FUNCTION_BLOCK FB_FallibleSTRINGMock IMPLEMENTS I_FallibleSTRING
VAR
    bError : BOOL;
    sErrorMsg : T_MaxString;
    sVal : STRING;
END_VAR


METHOD ClearError

bError := FALSE;
sErrorMsg := '';
END_METHOD


METHOD GetError : BOOL

GetError := THIS^.bError;
END_METHOD


METHOD GetErrorMsg : T_MaxString

GetErrorMsg := sErrorMsg;
END_METHOD


METHOD PUBLIC SetError
VAR_INPUT
    sMsg : T_MaxString;
END_VAR

THIS^.bError := TRUE;
END_METHOD


PROPERTY Val : STRING
GET

Val := THIS^.sVal;
END_GET
SET

THIS^.sVal := Val;
END_SET
END_PROPERTY

END_FUNCTION_BLOCK

(* stored: Version 1.1.0.1
   POU FB_FallibleSTRINGMock: Id {a03a76bb-b88e-4cb0-a83d-4c8c1047d27e}, SpecialFunc None
   Method ClearError: Id {5f0d1759-c39f-43fb-81f4-fdc5cc2e485e}
   Method GetError: Id {38ca86ff-2d69-45c3-8594-a73752ab4059}
   Method GetErrorMsg: Id {ed58391c-d097-418c-941e-d03465d9e920}
   Method SetError: Id {15147a93-ee16-439c-83ed-2024b54a6dad}
   Property Val: Id {be0a0c1c-d88a-43b9-9c51-e47d30841c5b}
   Get Get: Id {3c3643f5-c741-43d4-b826-94ecefd2c33e}
   Set Set: Id {1210e796-57a7-4707-93d8-7d3ef71a8b22} *)
